// TIA Portal project "2 Tetikleme ile Sıralı Çalıştırma Uygulaması_2" (V18)

(* hardware
DEVICE "S7-1200 station_1"  S7-1200 Station
   slot 0: "Rack_0"  S7-1200 Rack  Rack  V1.0
   slot 1: "PLC_1"  CPU 1214C AC/DC/Rly  6ES7 214-1BG40-0XB0  V4.6
*)

// ===== PLC "PLC_1"  CPU 1214C AC/DC/Rly =====

VAR_GLOBAL   // PLC tag table "Default tag table"
   "Stop" AT %I0.0 : Bool;
   "PKT_1" AT %I0.1 : Bool;
   "PKT_2" AT %I0.2 : Bool;
   "PKT_Yardımcı_1" AT %M0.0 : Bool;
   "Motor_1" AT %Q0.0 : Bool;
   "PKT_Yardımcı_2" AT %M0.1 : Bool;
   "PKT_3" AT %I0.3 : Bool;
   "PKT_Yardımcı_3" AT %M0.2 : Bool;
   "Tag_1" AT %Q0.1 : Bool;
   "Tag_2" AT %Q0.2 : Bool;
   "Tag_3" AT %M0.3 : Bool;
   "Tag_4" AT %M0.4 : Bool;
END_VAR

ORGANIZATION_BLOCK "Main"   // OB1, LAD, ProgramCycle
TITLE = "Main Program Sweep (Cycle)"
{ S7_Optimized_Access := 'TRUE' }
VERSION : 0.1
// *Bir tezgahta 2 adet motor çalıştırılacaktır. 
// *Start butonuna ilk kez basıldığında 1.motor çalışacak ve sürekli devrede kalacaktır. 
// *Start butonundan elimizi çektiğimiz anda 2. motor devreye girecek ve sürekli çalışacaktır. 
// *2 motor birlikte sürekli çalışırken durdurma butonuna basıldığı anda 2. motor duracak, durdurma butonundan elimizi çektiğimizde 1. motor duracaktır.
   VAR_INPUT
      Initial_Call : Bool;   // Initial call of this OB
      Remanence : Bool;   // =True, if remanent data are available
   END_VAR
   VAR_TEMP   // added for the SCL form of the ladder/FBD networks
      _w1 : Bool;
      _w2 : Bool;
      _w3 : Bool;
      _w4 : Bool;
   END_VAR
BEGIN

REGION Network 1
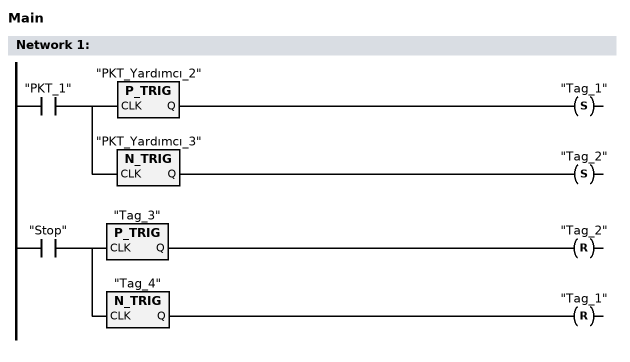
   RUNG wire#powerrail
      Contact( "PKT_1" )
      wire#w1
      P_Trig( "PKT_Yardımcı_2" )
      S_Coil( "Tag_1" )
   END_RUNG
   RUNG wire#w1
      N_Trig( "PKT_Yardımcı_3" )
      S_Coil( "Tag_2" )
   END_RUNG
   RUNG wire#powerrail
      Contact( "Stop" )
      wire#w2
      P_Trig( "Tag_3" )
      R_Coil( "Tag_2" )
   END_RUNG
   RUNG wire#w2
      N_Trig( "Tag_4" )
      R_Coil( "Tag_1" )
   END_RUNG
   // the same network as SCL:
   #_w1 := "PKT_1" AND NOT "PKT_Yardımcı_2";   // rising edge
   "PKT_Yardımcı_2" := "PKT_1";
   IF #_w1 THEN "Tag_1" := TRUE; END_IF;
   #_w2 := NOT "PKT_1" AND "PKT_Yardımcı_3";   // falling edge
   "PKT_Yardımcı_3" := "PKT_1";
   IF #_w2 THEN "Tag_2" := TRUE; END_IF;
   #_w3 := "Stop" AND NOT "Tag_3";   // rising edge
   "Tag_3" := "Stop";
   IF #_w3 THEN "Tag_2" := FALSE; END_IF;
   #_w4 := NOT "Stop" AND "Tag_4";   // falling edge
   "Tag_4" := "Stop";
   IF #_w4 THEN "Tag_1" := FALSE; END_IF;
END_REGION
END_ORGANIZATION_BLOCK